// TIA Portal V19 export
DATA_BLOCK "IPC_Com_Channel_LOG_PARAMETRI"   // DB222
// stored: MemoryReserve 100
   VAR
      RECEIVE : Struct   // Ricezione singolo messaggio da MES
         ack : DInt;   // Acknowledge msg.ID to MES
         msg : "IPC_Msg_Log_PAR";
      END_STRUCT;
      SEND : Struct   // Invio singolo messaggio a MES
         ack : DInt;   // Acknowledge msg.ID From MES
         msg : "IPC_Msg_Log_PAR";
      END_STRUCT;
   END_VAR
BEGIN
END_DATA_BLOCK
